# EPICS autosave request: BKHOFF/iocBoot/iocBKHOFF-IOC-01/BKHOFF_01_settings.req
# Motor settings
file "motor_settings.req" P=$(P),M=MTR$(CCP)01
file "motor_settings.req" P=$(P),M=MTR$(CCP)02
